ST1_ProductionDataValues:=	 CONCAT( ST1_ProductionDataValues,stStation1_ProductionData.DefaultNettWeight);
ST1_ProductionDataValues:= CONCAT( ST1_ProductionDataValues,',');
ST1_ProductionDataValues:=	 CONCAT( ST1_ProductionDataValues,stStation1_ProductionData.DefaultGrossWeight);
ST1_ProductionDataValues:= CONCAT( ST1_ProductionDataValues,',');
ST1_ProductionDataValues:=	 CONCAT( ST1_ProductionDataValues,stStation1_ProductionData.Blend);
ST1_ProductionDataValues:= CONCAT( ST1_ProductionDataValues,',');
ST1_ProductionDataValues:=	 CONCAT( ST1_ProductionDataValues,stStation1_ProductionData.Shade);
ST1_ProductionDataValues:= CONCAT( ST1_ProductionDataValues,',');
ST1_ProductionDataValues:=	 CONCAT( ST1_ProductionDataValues,stStation1_ProductionData.ConeTip);
ST1_ProductionDataValues:= CONCAT( ST1_ProductionDataValues,',');
ST1_ProductionDataValues:=	 CONCAT( ST1_ProductionDataValues,stStation1_ProductionData.ConeNettWeight);
ST1_ProductionDataValues:= CONCAT( ST1_ProductionDataValues,',');
ST1_ProductionDataValues:=	 CONCAT( ST1_ProductionDataValues,stStation1_ProductionData.ConeLength);
ST1_ProductionDataValues:= CONCAT( ST1_ProductionDataValues,',');
ST1_ProductionDataValues:=	 CONCAT( ST1_ProductionDataValues,stStation1_ProductionData.Dom_Exp);
ST1_ProductionDataValues:= CONCAT( ST1_ProductionDataValues,',');
ST1_ProductionDataValues:=	 CONCAT( ST1_ProductionDataValues,stStation1_ProductionData.PackType);
ST1_ProductionDataValues:= CONCAT( ST1_ProductionDataValues,',');
ST1_ProductionDataValues:=	 CONCAT( ST1_ProductionDataValues,stStation1_ProductionData.CountCode);
ST1_ProductionDataValues:= CONCAT( ST1_ProductionDataValues,'$0A');
(*==========Saving the Data to Report===========*)


sStation1_ProductionData_FileName:= Fb_CreateFileFormat_1.sOldFileName ; (*    'Hard Disk\Reports\Test1\ProductionData.csv' ;*)


Fb_LoagProductionData(
	bStartDataLog:= SaveData ,
	sDataLogFileName:=sStation1_ProductionData_FileName ,
	LogData:=ST1_ProductionDataValues ,
	bErrorDataLog=> );






(*=============== file copy from CX Controller to Remote PC & File Delete In CX Device======================*)


	Fb_CopyBackupAL_Server_LogOf_1(
		bMakeDirectory:= ,
		bCopyFile:=bool2,
		sDestDriveName:=' \\Admin-PC\Public\',
		sSourceDirectory:='\Hard Disk\Reports\Indo' ,
		 );

(*\\ramrajg-nb2\Ramaraj_public\   *)

  (*Hard Disk\Reports\  *)

Fb_FormatDrive_1(sDriveName:= '\\Admin-PC\Public\', bFormatDisk:=bFileDelete );

R_TRIG1(CLK:=CycleComplete OR CycleComplete1 , Q=> );


CASE ReportStep OF

	0:	 IF R_TRIG1.Q   THEN  FileCreateTemp:=TRUE; Timer3(IN:=FALSE); ReportStep:=1; END_IF

	1:	(*		##### Station 1 Production Data	#####	*)

		ST1_ProductionData:= CONCAT( 'S.No',',');
		ST1_ProductionData:=	 CONCAT( ST1_ProductionData,'Cone Type');
		ST1_ProductionData:= CONCAT( ST1_ProductionData,',');
		ST1_ProductionData:=	 CONCAT( ST1_ProductionData,'Carton No');
		ST1_ProductionData:= CONCAT( ST1_ProductionData,',');
		ST1_ProductionData:=	 CONCAT( ST1_ProductionData,'Lot No');
		ST1_ProductionData:= CONCAT( ST1_ProductionData,',');
		ST1_ProductionData:=	 CONCAT( ST1_ProductionData,'Date');
		ST1_ProductionData:= CONCAT( ST1_ProductionData,',');
		ST1_ProductionData:=	 CONCAT( ST1_ProductionData,'Net Weight');
		ST1_ProductionData:= CONCAT( ST1_ProductionData,',');
		ST1_ProductionData:=	 CONCAT( ST1_ProductionData,'Work Order No');
		ST1_ProductionData:= CONCAT( ST1_ProductionData,',');

ST1_ProductionData:=	 CONCAT( ST1_ProductionData,'Default Net Weight');
		ST1_ProductionData:= CONCAT( ST1_ProductionData,',');
ST1_ProductionData:=	 CONCAT( ST1_ProductionData,'Defaulr Gross Weight');
		ST1_ProductionData:= CONCAT( ST1_ProductionData,',');
ST1_ProductionData:=	 CONCAT( ST1_ProductionData,'Blend');
		ST1_ProductionData:= CONCAT( ST1_ProductionData,',');
ST1_ProductionData:=	 CONCAT( ST1_ProductionData,'Shade');
		ST1_ProductionData:= CONCAT( ST1_ProductionData,',');
ST1_ProductionData:=	 CONCAT( ST1_ProductionData,'Cone Tip');
		ST1_ProductionData:= CONCAT( ST1_ProductionData,',');
ST1_ProductionData:=	 CONCAT( ST1_ProductionData,'Cone Nett Weight');
		ST1_ProductionData:= CONCAT( ST1_ProductionData,',');
ST1_ProductionData:=	 CONCAT( ST1_ProductionData,'Cone Length');
		ST1_ProductionData:= CONCAT( ST1_ProductionData,',');
ST1_ProductionData:=	 CONCAT( ST1_ProductionData,'Dom Exp');
		ST1_ProductionData:= CONCAT( ST1_ProductionData,',');
ST1_ProductionData:=	 CONCAT( ST1_ProductionData,'Pack Type');
		ST1_ProductionData:=CONCAT( ST1_ProductionData,',');
ST1_ProductionData:=	 CONCAT( ST1_ProductionData,'CountCode');
		ST1_ProductionData:= CONCAT( ST1_ProductionData,'$0A');
		ReportStep:=2;

	2:	Timer1(IN:=FALSE);
		bANewDay:=FALSE;
		ReportStep:=3;


	3:	bEnableFileFormat:=TRUE;
		Timer1(IN:=TRUE , PT:=T#100ms , Q=> , ET=> );
		IF Timer1.Q THEN bEnableFileFormat:=FALSE;  ReportStep:=4; END_IF


	4:
		SaveData:=TRUE;
		Timer1(IN:=FALSE);
		ReportStep:=5;

	5:	Timer3(IN:=TRUE , PT:=T#25s , Q=> , ET=> );
		IF Timer3.Q THEN SaveData:=FALSE;bFileDelete:=TRUE; ReportStep:=6; END_IF

	6:	 bFileDelete:=FALSE;Timer3(IN:=FALSE); FileCreateTemp:=FALSE; ReportStep:=0;

END_CASE





IF ParametesSave THEN LotNoChange:=TRUE;ELSE LotNoChange:=FALSE;END_IF

IF bAutoModeOn AND bAPauseSeq AND   LotNoChange  THEN
	CurrentCartonNo:=CartonNoHmi;LotChangeCompleted:=FALSE;SameLotNo:=FALSE;
 END_IF

IF bAutoModeOn AND LotChangeCompleted THEN
	iLotNoPrevious:=iLotNoHmi;
END_IF



IF iLotNoPrevious=iLotNoHmi THEN SameLotNo:=TRUE;
ELSE SameLotNo:=FALSE;END_IF

CASE CartonNo OF

0: 	IF (CycleComplete OR CycleComplete1) THEN CartonNo:=CartonNo+1;TON_CountCheck(IN:=FALSE);END_IF

1:	IF SameLotNo THEN CartonNo:=CartonNo+1;
	ELSIF NOT SameLotNo THEN CartonNo:=3;END_IF

2:	CurrentCartonNo:=CurrentCartonNo+1;CartonNo:=4;

3:	CurrentCartonNo:=CartonNoHmi;CartonNo:=CartonNo+1;

4:	TON_CountCheck(IN:=TRUE, PT:=t#30s, Q=> , ET=> );
	IF TON_CountCheck.Q THEN CartonNo:=CartonNo+1;END_IF

5:	CartonNo:=0;LotChangeCompleted:=TRUE;

END_CASE









(*
CASE StepTemp1 OF
	0:	IF bRetUnitBStart THEN rRetUnitBWeightTemp1:=rRetUnitBWeight; StepTemp1:=StepTemp1+1; END_IF

	1:	IF UnitBCompleteCheckCount.CV = 18 AND bAutoModeOn THEN rRetUnitBWeightTemp2:=rRetUnitBWeightTemp1;  StepTemp1:=0; END_IF
 END_CASE




CASE StepTemp2 OF
	0:	IF bRetUnitBStart THEN rRetUnitBWeightTemp1:=rRetUnitBWeight; StepTemp2:=StepTemp2+1; END_IF

	1:	IF c18_ConeCounter1.CV = 18 AND bAutoModeOn THEN rRetUnitBWeightTemp2:=rRetUnitBWeightTemp1; c18_ConeCounter1.RESET:=TRUE;  StepTemp2:=StepTemp2+1; END_IF

	2:	c18_ConeCounter1.RESET:=FALSE;  StepTemp2:=0;
 END_CASE*)


(*IF LotAHmi AND NOT LotBHmi AND NOT LotCHmi THEN LotASelected:=TRUE;LotBSelected:=FALSE;LotCSelected:=FALSE;END_IF
IF NOT LotAHmi AND  LotBHmi AND NOT LotCHmi THEN LotBSelected:=TRUE;LotASelected:=FALSE;LotCSelected:=FALSE;END_IF
IF NOT LotAHmi AND NOT LotBHmi AND  LotCHmi THEN LotCSelected:=TRUE;LotBSelected:=FALSE;LotASelected:=FALSE;END_IF

IF LotASelected THEN CartonNoHmi:=LotACartonNo;
ELSIF LotBSelected THEN CartonNoHmi:=LotBCartonNo;
ELSIF  LotCSelected THEN CartonNoHmi:=LotCCartonNo;
ELSIF  LotDSelected THEN CartonNoHmi:=LotDCartonNo;
ELSIF  LotESelected THEN CartonNoHmi:=LotECartonNo;
ELSIF  LotFSelected THEN CartonNoHmi:=LotFCartonNo;
END_IF

IF CartonNoResetHmi OR  (NOT LotAHmi AND NOT LotBHmi AND NOT LotCHmi) THEN
	LotACartonNo:=0;
	LotBCartonNo:=0;
	LotCCartonNo:=0;
	LotDCartonNo:=0;
	LotECartonNo:=0;
	LotFCartonNo:=0;
END_IF



CASE LotA OF

0:	IF LotASelected THEN LotA:=LotA+1;END_IF

1:	IF (CycleComplete OR CycleComplete1) THEN LotA :=LotA +1;END_IF

2:	LotACartonNo:=LotACartonNo+1;
	LotA :=LotA +1;

3:	TON_11(IN:=TRUE , PT:=t#25s , Q=> , ET=> );
	IF TON_11.Q THEN LotA :=LotA +1;END_IF

4:	LotA :=0;

END_CASE


CASE LotB OF

0:	IF LotBSelected THEN LotB:=LotB+1;END_IF

1:	IF (CycleComplete OR CycleComplete1) THEN LotB:=LotB+1;END_IF

2:	LotBCartonNo:=LotBCartonNo+1;
	LotB:=LotB+1;

3:	TON_12(IN:=TRUE , PT:=t#25s , Q=> , ET=> );
	IF TON_12.Q THEN LotA :=LotA +1;END_IF

4:	LotB:=0;

END_CASE


CASE LotC OF

0:	IF LotCSelected THEN LotC:=LotC+1;END_IF

1:	IF (CycleComplete OR CycleComplete1) THEN LotC:=LotC+1;END_IF

2:	LotCCartonNo:=LotCCartonNo+1;
	LotC:=LotC+1;

3:	TON_13(IN:=TRUE , PT:=t#25s , Q=> , ET=> );
	IF TON_13.Q THEN LotA :=LotA +1;END_IF

4:	LotC:=0;

END_CASE*)
END_PROGRAM

(* POU FunctionBlocks/DATA_LOG_Save, ST *)
FUNCTION_BLOCK DATA_LOG_Save
VAR_INPUT
	bStartDataLog: BOOL;
	sDataLogFileName: STRING;
	LogData: STRING(1024);

END_VAR
VAR_OUTPUT

	bErrorDataLog: BOOL;
END_VAR
VAR

	R_TRIGStartDataLog: R_TRIG;
	nstep: INT;

	FB_OpenFile_Datalog: FB_FileOpen;
	nFB_OpenFile_Datalog_Errid: UDINT;

	FB_WriteFile_Datalog: FB_FileWrite;
	nFB_WriteFile_Datalog_ErrId: UDINT;

	FB_CloseFile_Datalog: FB_FileClose;
	nFB_CloseFile_Datalog_ErrId: UDINT;
	hDataLogSrcFile: UINT;

END_VAR
R_TRIGStartDataLog(CLK:=bStartDataLog , Q=> );
IF R_TRIGStartDataLog.Q THEN
		nstep :=1;
	END_IF

CASE nstep OF

	0:
		;
		FB_OpenFile_Datalog.bExecute:=FALSE;
		FB_WriteFile_Datalog.bExecute:=FALSE;
		FB_CloseFile_Datalog.bExecute:=FALSE;

	1:		(* do nothing *)
			nstep:=nstep+1;

	2:		(* ####	File Open ####*)

			FB_OpenFile_Datalog(  bExecute := FALSE  );
			FB_OpenFile_Datalog(	sNetId :='192.168.0.103.1.1' ,
			sPathName := sDataLogFileName,
			nMode := FOPEN_MODEAPPEND    ,
			ePath := PATH_GENERIC,
			tTimeout := T#2s,
			bExecute := TRUE );
			nstep := nstep+ 1;



	3:		FB_OpenFile_Datalog( bExecute := FALSE );
			IF ( NOT FB_OpenFile_Datalog.bBusy ) THEN
			IF ( FB_OpenFile_Datalog.bError ) THEN
			nFB_OpenFile_Datalog_Errid := FB_OpenFile_Datalog.nErrId;
			bErrorDataLog := TRUE;
			nstep := 50;
			ELSE
			hDataLogSrcFile := FB_OpenFile_Datalog.hFile;
			nstep := nstep + 1;
			END_IF
			END_IF

	4:		(*write data to destination file*)
			(*num:=num+1;*)
			FB_WriteFile_Datalog( bExecute := FALSE );
			FB_WriteFile_Datalog(	sNetId:='192.168.0.103.1.1',
			hFile:=FB_OpenFile_Datalog.hFile,
			pWriteBuff:= ADR(LogData),
			cbWriteLen:= LEN(LogData),		(*	i_len,	*)
			bExecute:=TRUE,
			tTimeout:=T#2s );
			nstep := nstep + 1;

	5:		FB_WriteFile_Datalog( bExecute := FALSE );
			IF ( NOT FB_WriteFile_Datalog.bBusy ) THEN
			IF ( FB_WriteFile_Datalog.bError ) THEN
			nFB_WriteFile_Datalog_ErrId := FB_WriteFile_Datalog.nErrId;
			bErrorDataLog := TRUE;
			nstep := 50;
			ELSE
			hDataLogSrcFile := FB_OpenFile_Datalog.hFile;
			nstep := nstep + 1;
			END_IF
			END_IF

	6:		(* close the destination file *)
			FB_CloseFile_Datalog( bExecute := FALSE );
			FB_CloseFile_Datalog( 	sNetId:='192.168.0.103.1.1' ,
			hFile:=FB_OpenFile_Datalog.hFile,
			bExecute:=TRUE,
			tTimeout:=T#2s );
			nstep := nstep + 1;

	7:		FB_CloseFile_Datalog( bExecute := FALSE );
			IF ( NOT FB_CloseFile_Datalog.bBusy ) THEN
			IF ( FB_CloseFile_Datalog.bError ) THEN
			nFB_CloseFile_Datalog_ErrId := FB_CloseFile_Datalog.nErrId;
			bErrorDataLog := TRUE;
			END_IF
			nstep := 0;
			END_IF

END_CASE
END_FUNCTION_BLOCK

(* POU FunctionBlocks/Fb_CreateFileFormat, LD *)
FUNCTION_BLOCK Fb_CreateFileFormat
VAR
	Fb_OpenFile: FB_FileOpen;
	Fb_WriteFile: FB_FileWrite;
	F_Trig1: F_TRIG;
	F_Trig2: F_TRIG;
	Fb_closeFile: FB_FileClose;
	F_Trig3: F_TRIG;


	SysteMtime: FB_LocalSystemTime;
	stSystemtimeAlrm: Timestruct;

	sFileName_Temp: T_MaxString;


	bCreateFileTrig: R_TRIG;
	bCreateFile: BOOL;
	Fb_SavePersistant: FB_WritePersistentData;
	TuneparaSave: BOOL;
END_VAR
VAR_INPUT

	sInputMessage: STRING(255);
	sFileName: T_MaxString;
	sDirectory: T_MaxString;
	bEnable: BOOL;

END_VAR
VAR_OUTPUT

	sDate: STRING;

	bNewDateFound: BOOL;
END_VAR

VAR_OUTPUT PERSISTENT
	sOldFileName: T_MaxString;
	sFilePathFinal: t_MaxString;
END_VAR
VAR PERSISTENT
	sOldDate: STRING;
	sNewFileName_Temp: T_MaxString;
END_VAR
VAR_IN_OUT PERSISTENT
	wToday: STRING;
END_VAR
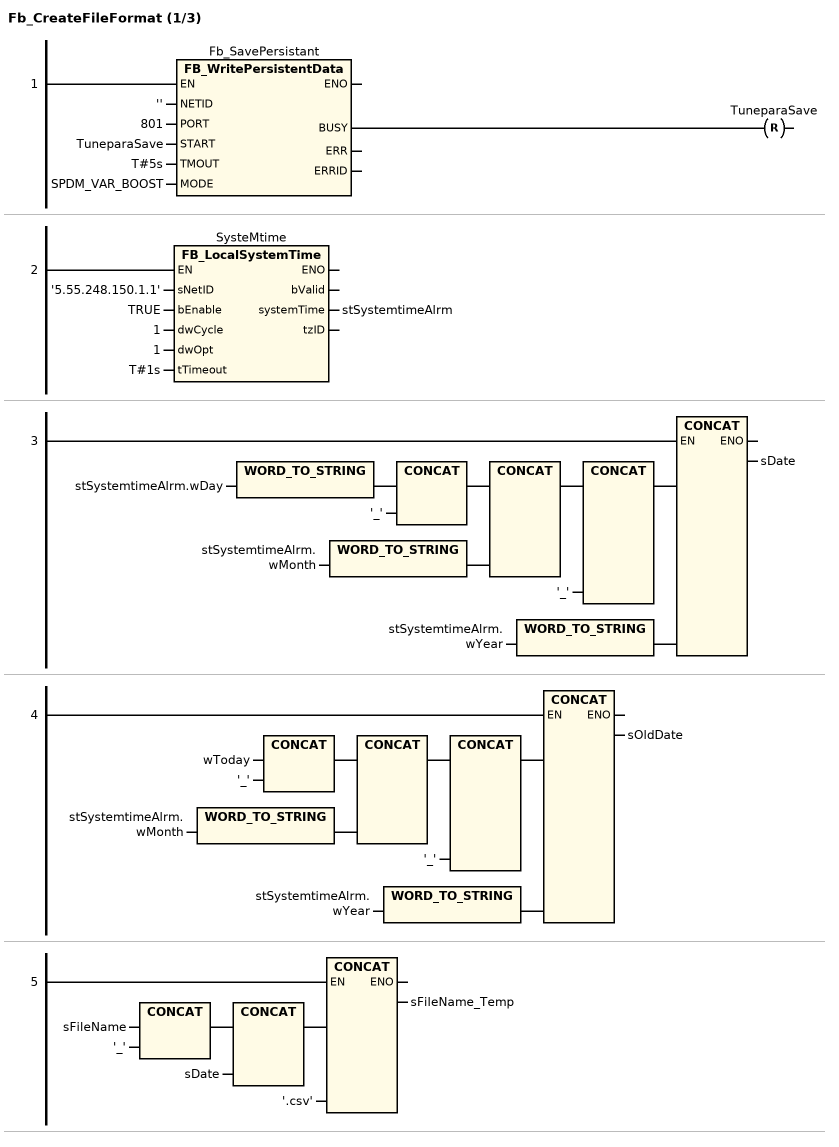
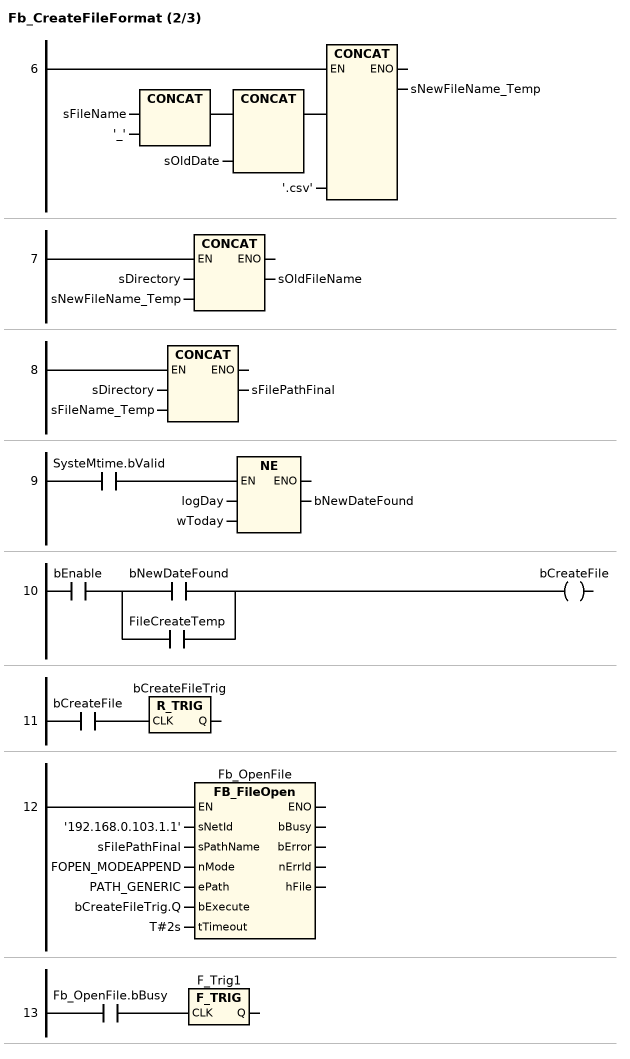
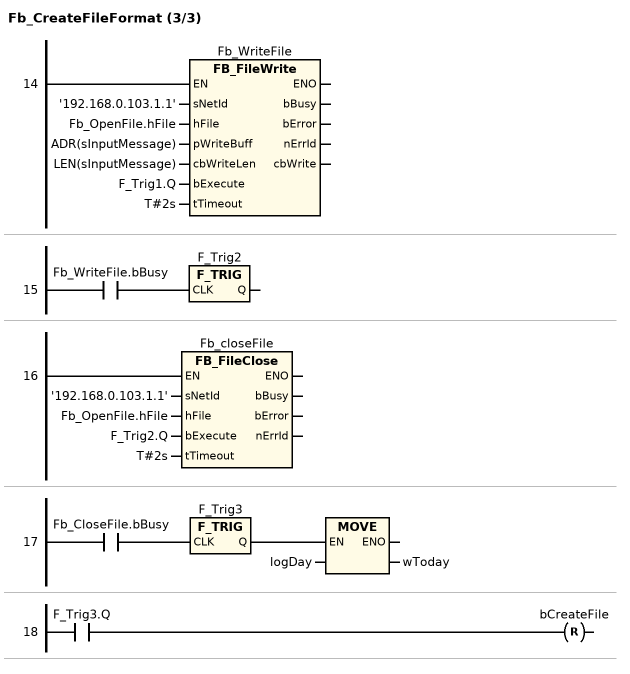
_LD_ (* Ladder Diagram *)
NETWORK 1
	*
		EN --- Fb_SavePersistant:FB_WritePersistentData(NETID: '', PORT: 801, START: TuneparaSave, TMOUT: T#5s, MODE: SPDM_VAR_BOOST) => R TuneparaSave
NETWORK 2
	*
		EN --- SysteMtime:FB_LocalSystemTime(sNetID: '5.55.248.150.1.1', bEnable: TRUE, dwCycle: 1, dwOpt: 1, tTimeout: T#1s, systemTime => stSystemtimeAlrm)
NETWORK 3
	*
		EN --- CONCAT(CONCAT(CONCAT(CONCAT(WORD_TO_STRING(stSystemtimeAlrm.wDay), '_'), WORD_TO_STRING(stSystemtimeAlrm.wMonth)), '_'), WORD_TO_STRING(stSystemtimeAlrm.wYear)) => sDate
NETWORK 4
	*
		EN --- CONCAT(CONCAT(CONCAT(CONCAT(wToday, '_'), WORD_TO_STRING(stSystemtimeAlrm.wMonth)), '_'), WORD_TO_STRING(stSystemtimeAlrm.wYear)) => sOldDate
NETWORK 5
	*
		EN --- CONCAT(CONCAT(CONCAT(sFileName, '_'), sDate), '.csv') => sFileName_Temp
NETWORK 6
	*
		EN --- CONCAT(CONCAT(CONCAT(sFileName, '_'), sOldDate), '.csv') => sNewFileName_Temp
NETWORK 7
	*
		EN --- CONCAT(sDirectory, sNewFileName_Temp) => sOldFileName
NETWORK 8
	*
		EN --- CONCAT(sDirectory, sFileName_Temp) => sFilePathFinal
NETWORK 9
	[SysteMtime.bValid]
		EN --- NE(logDay, wToday) => bNewDateFound
NETWORK 10
	[bEnable] - { [bNewDateFound] | [FileCreateTemp] } --- (bCreateFile)
NETWORK 11
	[bCreateFile] - bCreateFileTrig:R_TRIG(CLK: *)
NETWORK 12
	*
		EN --- Fb_OpenFile:FB_FileOpen(sNetId: '192.168.0.103.1.1', sPathName: sFilePathFinal, nMode: FOPEN_MODEAPPEND, ePath: PATH_GENERIC, bExecute: bCreateFileTrig.Q, tTimeout: T#2s)
NETWORK 13
	[Fb_OpenFile.bBusy] - F_Trig1:F_TRIG(CLK: *)
NETWORK 14
	*
		EN --- Fb_WriteFile:FB_FileWrite(sNetId: '192.168.0.103.1.1', hFile: Fb_OpenFile.hFile, pWriteBuff: ADR(sInputMessage), cbWriteLen: LEN(sInputMessage), bExecute: F_Trig1.Q, tTimeout: T#2s)
NETWORK 15
	[Fb_WriteFile.bBusy] - F_Trig2:F_TRIG(CLK: *)
NETWORK 16
	*
		EN --- Fb_closeFile:FB_FileClose(sNetId: '192.168.0.103.1.1', hFile: Fb_OpenFile.hFile, bExecute: F_Trig2.Q, tTimeout: T#2s)
NETWORK 17
	[Fb_CloseFile.bBusy] - F_Trig3:F_TRIG(CLK: *)
		EN --- MOVE(logDay) => wToday
NETWORK 18
	[F_Trig3.Q] --- (R bCreateFile)
_END_LD_
(* the same logic as Structured Text *)
(* Network 1 *)
Fb_SavePersistant(NETID := '', PORT := 801, START := TuneparaSave, TMOUT := T#5s, MODE := SPDM_VAR_BOOST);
IF Fb_SavePersistant.BUSY THEN TuneparaSave := FALSE; END_IF;
(* Network 2 *)
SysteMtime(sNetID := '5.55.248.150.1.1', bEnable := TRUE, dwCycle := 1, dwOpt := 1, tTimeout := T#1s);
stSystemtimeAlrm := SysteMtime.systemTime;
(* Network 3 *)
sDate := CONCAT(CONCAT(CONCAT(CONCAT(WORD_TO_STRING(stSystemtimeAlrm.wDay), '_'), WORD_TO_STRING(stSystemtimeAlrm.wMonth)), '_'), WORD_TO_STRING(stSystemtimeAlrm.wYear));
(* Network 4 *)
sOldDate := CONCAT(CONCAT(CONCAT(CONCAT(wToday, '_'), WORD_TO_STRING(stSystemtimeAlrm.wMonth)), '_'), WORD_TO_STRING(stSystemtimeAlrm.wYear));
(* Network 5 *)
sFileName_Temp := CONCAT(CONCAT(CONCAT(sFileName, '_'), sDate), '.csv');
(* Network 6 *)
sNewFileName_Temp := CONCAT(CONCAT(CONCAT(sFileName, '_'), sOldDate), '.csv');
(* Network 7 *)
sOldFileName := CONCAT(sDirectory, sNewFileName_Temp);
(* Network 8 *)
sFilePathFinal := CONCAT(sDirectory, sFileName_Temp);
(* Network 9 *)
IF SysteMtime.bValid THEN
	bNewDateFound := logDay <> wToday;
END_IF;
(* Network 10 *)
bCreateFile := bEnable AND (bNewDateFound OR FileCreateTemp);
(* Network 11 *)
bCreateFileTrig(CLK := bCreateFile);
(* Network 12 *)
Fb_OpenFile(sNetId := '192.168.0.103.1.1', sPathName := sFilePathFinal, nMode := FOPEN_MODEAPPEND, ePath := PATH_GENERIC, bExecute := bCreateFileTrig.Q, tTimeout := T#2s);
(* Network 13 *)
F_Trig1(CLK := Fb_OpenFile.bBusy);
(* Network 14 *)
Fb_WriteFile(sNetId := '192.168.0.103.1.1', hFile := Fb_OpenFile.hFile, pWriteBuff := ADR(sInputMessage), cbWriteLen := LEN(sInputMessage), bExecute := F_Trig1.Q, tTimeout := T#2s);
(* Network 15 *)
F_Trig2(CLK := Fb_WriteFile.bBusy);
(* Network 16 *)
Fb_closeFile(sNetId := '192.168.0.103.1.1', hFile := Fb_OpenFile.hFile, bExecute := F_Trig2.Q, tTimeout := T#2s);
(* Network 17 *)
F_Trig3(CLK := Fb_CloseFile.bBusy);
IF F_Trig3.Q THEN
	wToday := logDay;
END_IF;
(* Network 18 *)
IF F_Trig3.Q THEN bCreateFile := FALSE; END_IF;
END_FUNCTION_BLOCK

(* POU AutoMode/Fb_FormatDrive, FBD *)
FUNCTION_BLOCK Fb_FormatDrive
VAR_INPUT
	sDriveName: T_MaxString;
	bFormatDisk: BOOL;
END_VAR
VAR_OUTPUT
END_VAR
VAR
	sDeleteCommand_Temp: T_MaxString;
	sDeleteCommand: T_MaxString;
	nDirectoryLength: INT;
	sFormatedDirectory: T_MaxString;
	FbFormatDisk: NT_StartProcess;
END_VAR
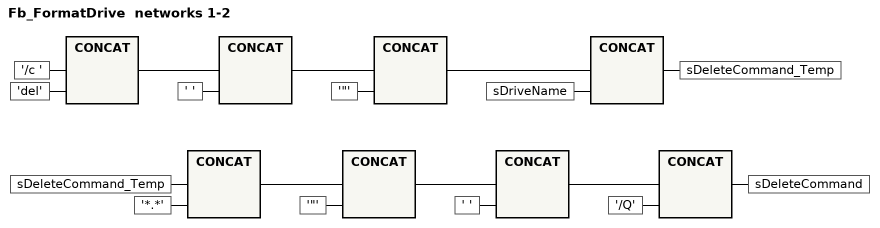
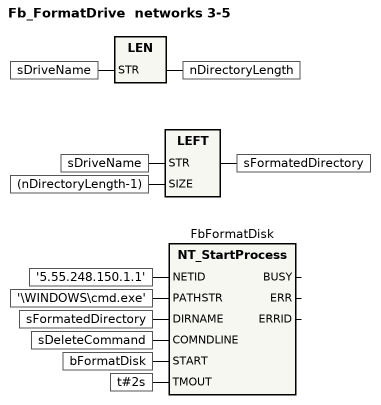
_FBD_ (* Function Block Diagram *)
NETWORK 1
	CONCAT(CONCAT(CONCAT(CONCAT('/c ', 'del'), ' '), '"'), sDriveName) => sDeleteCommand_Temp
NETWORK 2
	CONCAT(CONCAT(CONCAT(CONCAT(sDeleteCommand_Temp, '*.*'), '"'), ' '), '/Q') => sDeleteCommand
NETWORK 3
	LEN(STR: sDriveName) => nDirectoryLength
NETWORK 4
	LEFT(STR: sDriveName, SIZE: (nDirectoryLength-1)) => sFormatedDirectory
NETWORK 5
	FbFormatDisk:NT_StartProcess(NETID: '5.55.248.150.1.1', PATHSTR: '\WINDOWS\cmd.exe', DIRNAME: sFormatedDirectory, COMNDLINE: sDeleteCommand, START: bFormatDisk, TMOUT: t#2s)
_END_FBD_
(* the same logic as Structured Text *)
(* Network 1 *)
sDeleteCommand_Temp := CONCAT(CONCAT(CONCAT(CONCAT('/c ', 'del'), ' '), '"'), sDriveName);
(* Network 2 *)
sDeleteCommand := CONCAT(CONCAT(CONCAT(CONCAT(sDeleteCommand_Temp, '*.*'), '"'), ' '), '/Q');
(* Network 3 *)
nDirectoryLength := LEN(sDriveName);
(* Network 4 *)
sFormatedDirectory := LEFT(sDriveName, (nDirectoryLength-1));
(* Network 5 *)
FbFormatDisk(NETID := '5.55.248.150.1.1', PATHSTR := '\WINDOWS\cmd.exe', DIRNAME := sFormatedDirectory, COMNDLINE := sDeleteCommand, START := bFormatDisk, TMOUT := t#2s);
END_FUNCTION_BLOCK

(* POU FunctionBlocks/Fb_CopyFileToRemotePC, FBD *)
FUNCTION_BLOCK Fb_CopyFileToRemotePC
VAR
	sCopyFileCommandTemp: T_MaxString;
	sFormatedDestDirectory: T_Maxstring;
	sCopyFileCommand: T_MaxString;
	sFormatedDirectory: T_MaxString;
	sMakeDirCommand: T_MaxString;

	Fb_SystemTime: FB_LocalSystemTime;
	FB_MakeDirectory: NT_StartProcess;
	Fb_CopyFiles: NT_StartProcess;
END_VAR
VAR_INPUT

	bMakeDirectory: BOOL;
	bCopyFile: BOOL;
	sDestDriveName: T_MaxString;
	sSourceDirectory: T_MaxString;
END_VAR
VAR_OUTPUT
	sFinalDestDirectory: T_MaxString;
END_VAR
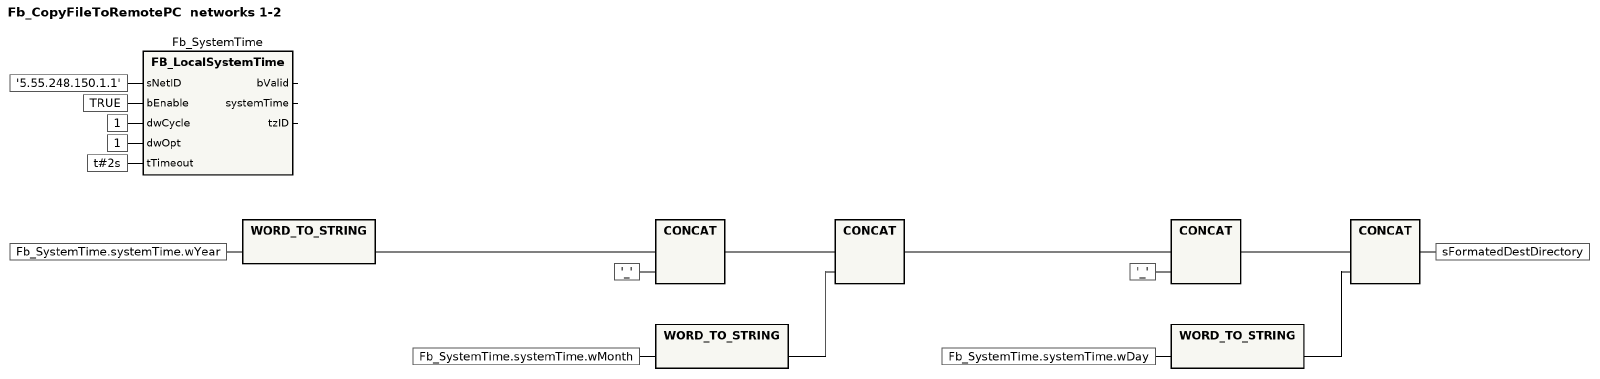
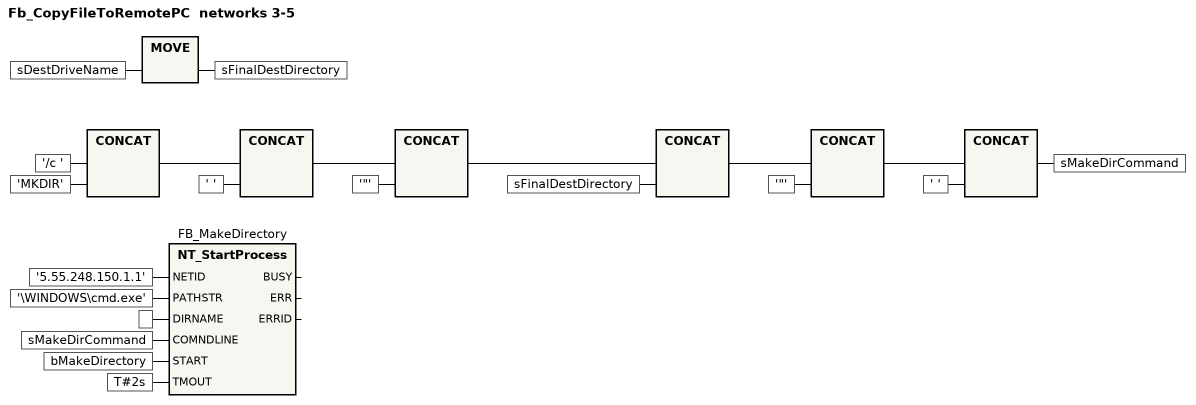
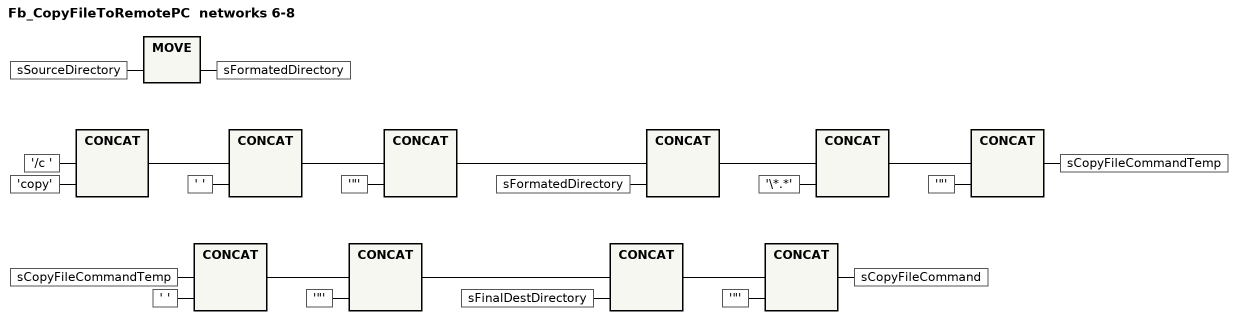
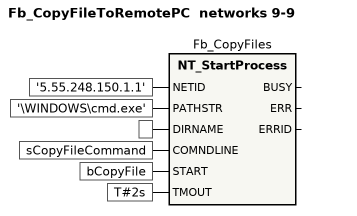
_FBD_ (* Function Block Diagram *)
NETWORK 1
	Fb_SystemTime:FB_LocalSystemTime(sNetID: '5.55.248.150.1.1', bEnable: TRUE, dwCycle: 1, dwOpt: 1, tTimeout: t#2s)
NETWORK 2
	CONCAT(CONCAT(CONCAT(CONCAT(WORD_TO_STRING(Fb_SystemTime.systemTime.wYear), '_'), WORD_TO_STRING(Fb_SystemTime.systemTime.wMonth)), '_'), WORD_TO_STRING(Fb_SystemTime.systemTime.wDay)) => sFormatedDestDirectory
NETWORK 3
	MOVE(sDestDriveName) => sFinalDestDirectory
NETWORK 4
	CONCAT(CONCAT(CONCAT(CONCAT(CONCAT(CONCAT('/c ', 'MKDIR'), ' '), '"'), sFinalDestDirectory), '"'), ' ') => sMakeDirCommand
NETWORK 5
	FB_MakeDirectory:NT_StartProcess(NETID: '5.55.248.150.1.1', PATHSTR: '\WINDOWS\cmd.exe', DIRNAME: , COMNDLINE: sMakeDirCommand, START: bMakeDirectory, TMOUT: T#2s)
NETWORK 6
	MOVE(sSourceDirectory) => sFormatedDirectory
NETWORK 7
	CONCAT(CONCAT(CONCAT(CONCAT(CONCAT(CONCAT('/c ', 'copy'), ' '), '"'), sFormatedDirectory), '\*.*'), '"') => sCopyFileCommandTemp
NETWORK 8
	CONCAT(CONCAT(CONCAT(CONCAT(sCopyFileCommandTemp, ' '), '"'), sFinalDestDirectory), '"') => sCopyFileCommand
NETWORK 9
	Fb_CopyFiles:NT_StartProcess(NETID: '5.55.248.150.1.1', PATHSTR: '\WINDOWS\cmd.exe', DIRNAME: , COMNDLINE: sCopyFileCommand, START: bCopyFile, TMOUT: T#2s)
_END_FBD_
(* the same logic as Structured Text *)
(* Network 1 *)
Fb_SystemTime(sNetID := '5.55.248.150.1.1', bEnable := TRUE, dwCycle := 1, dwOpt := 1, tTimeout := t#2s);
(* Network 2 *)
sFormatedDestDirectory := CONCAT(CONCAT(CONCAT(CONCAT(WORD_TO_STRING(Fb_SystemTime.systemTime.wYear), '_'), WORD_TO_STRING(Fb_SystemTime.systemTime.wMonth)), '_'), WORD_TO_STRING(Fb_SystemTime.systemTime.wDay));
(* Network 3 *)
sFinalDestDirectory := sDestDriveName;
(* Network 4 *)
sMakeDirCommand := CONCAT(CONCAT(CONCAT(CONCAT(CONCAT(CONCAT('/c ', 'MKDIR'), ' '), '"'), sFinalDestDirectory), '"'), ' ');
(* Network 5: see the listing above *)
(* Network 6 *)
sFormatedDirectory := sSourceDirectory;
(* Network 7 *)
sCopyFileCommandTemp := CONCAT(CONCAT(CONCAT(CONCAT(CONCAT(CONCAT('/c ', 'copy'), ' '), '"'), sFormatedDirectory), '\*.*'), '"');
(* Network 8 *)
sCopyFileCommand := CONCAT(CONCAT(CONCAT(CONCAT(sCopyFileCommandTemp, ' '), '"'), sFinalDestDirectory), '"');
(* Network 9: see the listing above *)
END_FUNCTION_BLOCK

(* Visualisation A
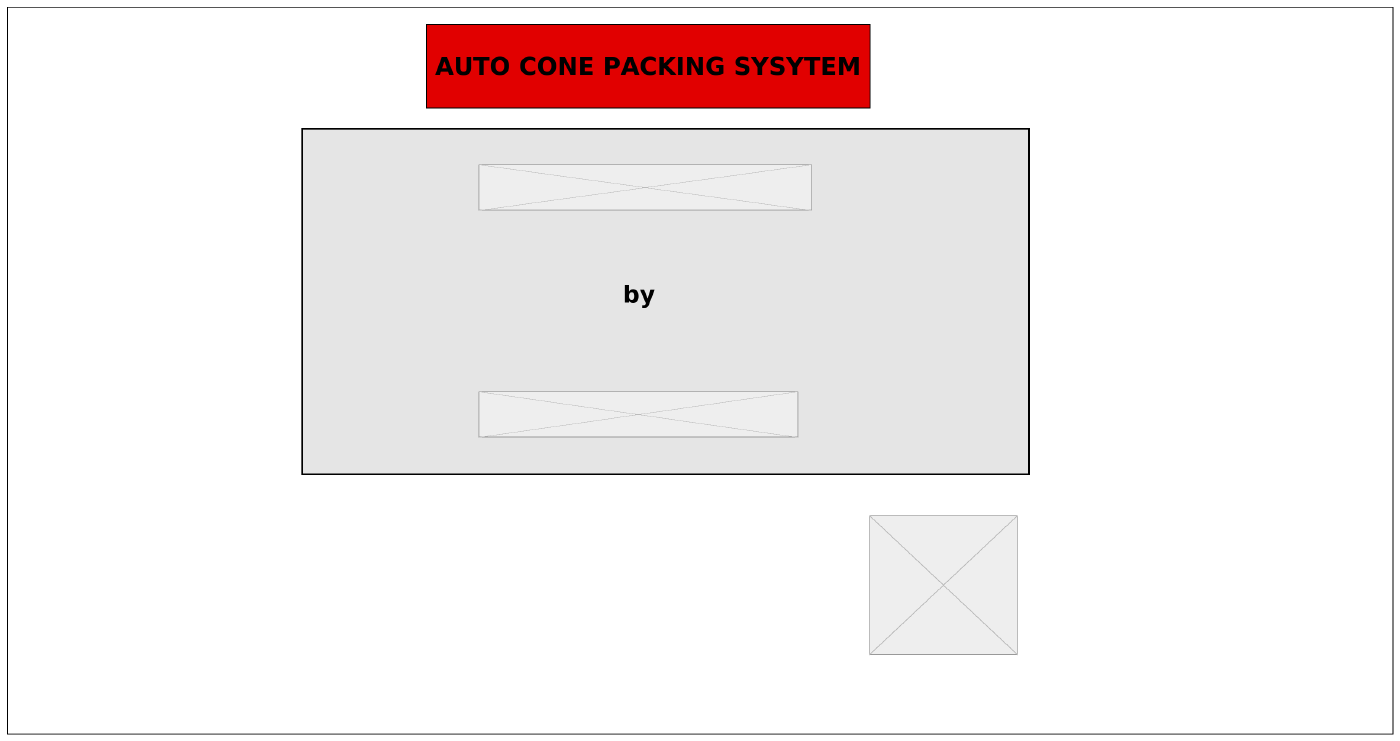
rounded rectangle at (484,20)-(997,117): text "AUTO CONE PACKING SYSYTEM"
bitmap at (996,588)-(1167,749): c:\twincat\plc\visu\startbutton.jpg
group at (340,140)-(1181,541)
  rounded rectangle at (0,0)-(1051,611): invisible if Common.EverRunTimer.Q
  bitmap at (256,64)-(737,145): c:\twincat\plc\visu\autocone-logom1.jpg
  bitmap at (256,464)-(717,545): c:\twincat\plc\visu\indo_logo1.bmp
  rectangle at (232,248)-(743,339): text "by"
2 more shapes without text or variables
*)

(* Visualisation ALARM
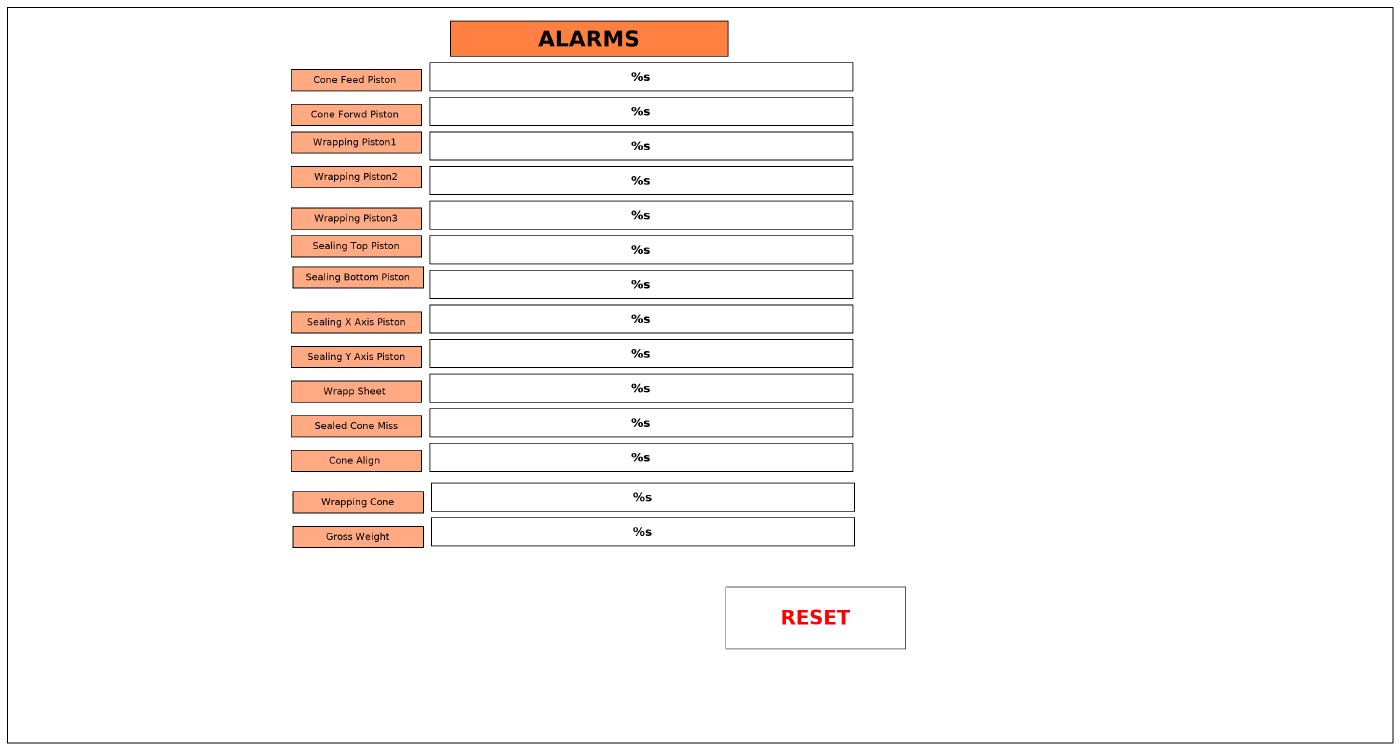
rounded rectangle at (328,112)-(479,137): text "Cone Forwd Piston"
rounded rectangle at (328,72)-(479,97): text "Cone Feed Piston"
rounded rectangle at (328,144)-(479,169): text "Wrapping Piston1"
rounded rectangle at (328,184)-(479,209): text "Wrapping Piston2"
rounded rectangle at (328,232)-(479,257): text "Wrapping Piston3"
rounded rectangle at (328,264)-(479,289): text "Sealing Top Piston"
rounded rectangle at (330,300)-(481,325): text "Sealing Bottom Piston"
rounded rectangle at (328,352)-(479,377): text "Sealing X Axis Piston"
rounded rectangle at (328,392)-(479,417): text "Sealing Y Axis Piston"
rectangle at (488,64)-(977,97): text "%s"; shows .HMIFeedPiston
rectangle at (488,224)-(977,257): text "%s"; shows .HMIWrapPiston3
rectangle at (488,184)-(977,217): text "%s"; shows .HMIWrapPiston2
rectangle at (488,264)-(977,297): text "%s"; shows .HMISealTopPiston
rectangle at (488,344)-(977,377): text "%s"; shows .HmiXAxisPiston
rectangle at (488,304)-(977,337): text "%s"; shows .HMISealBotPiston
rectangle at (488,384)-(977,417): text "%s"; shows .HmiYAxisPiston
rectangle at (488,144)-(977,177): text "%s"; shows .HMIWrapPiston1
rectangle at (488,104)-(977,137): text "%s"; shows .HMIForwdPiston
button at (830,670)-(1038,742): text "RESET"; shows .bErrorReset; taps .bErrorReset
rounded rectangle at (328,432)-(479,457): text "Wrapp Sheet"
rectangle at (488,424)-(977,457): text "%s"; shows ConeMissAlarm1
rounded rectangle at (328,472)-(479,497): text "Sealed Cone Miss"
rectangle at (488,464)-(977,497): text "%s"; shows .AlarmMessg
rounded rectangle at (328,512)-(479,537): text "Cone Align"
rectangle at (488,504)-(977,537): text "%s"; shows .ConeMissAlarm
rounded rectangle at (512,16)-(833,57): text "ALARMS"
rectangle at (490,550)-(979,583): text "%s"; shows WrapConeSenDetMes
rounded rectangle at (330,560)-(481,585): text "Wrapping Cone"
rectangle at (490,590)-(979,623): text "%s"; shows SGrossWtNokMsg
rounded rectangle at (330,600)-(481,625): text "Gross Weight"
1 more shapes without text or variables
2 elements of other kinds (tables, trends, ...) not read
*)

(* Visualisation ALARM_2
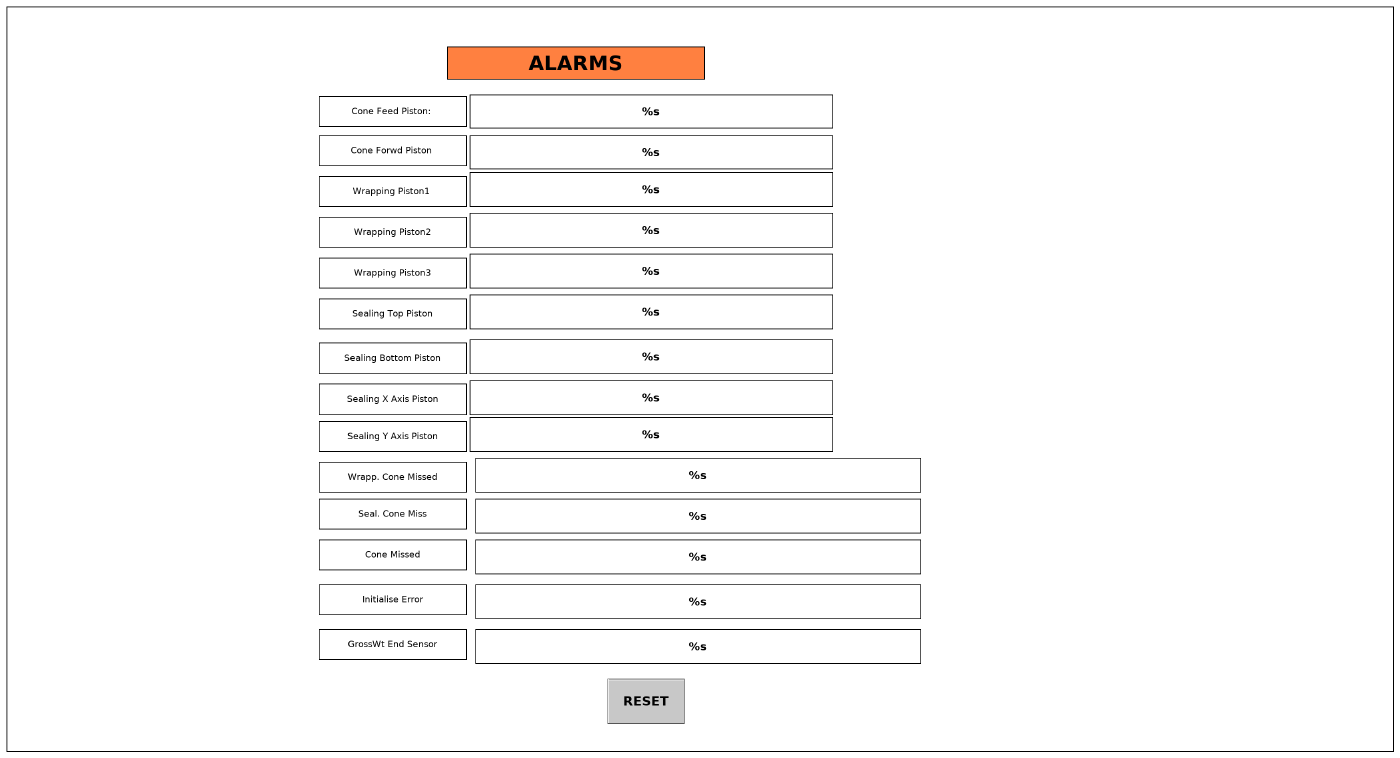
button at (750,830)-(846,886): text "RESET"; shows .bErrorReset; taps .bErrorReset
rounded rectangle at (550,40)-(871,81): text "ALARMS"
rounded rectangle at (390,151)-(574,189): text "Cone Forwd Piston"
rounded rectangle at (390,102)-(574,140): text "Cone Feed Piston:"
rounded rectangle at (390,202)-(574,240): text "Wrapping Piston1"
rounded rectangle at (390,253)-(574,291): text "Wrapping Piston2"
rounded rectangle at (390,304)-(574,342): text "Wrapping Piston3"
rounded rectangle at (390,355)-(574,393): text "Sealing Top Piston"
rounded rectangle at (390,410)-(574,449): text "Sealing Bottom Piston"
rounded rectangle at (390,461)-(574,500): text "Sealing X Axis Piston"
rounded rectangle at (390,508)-(574,546): text "Sealing Y Axis Piston"
rectangle at (578,100)-(1031,142): text "%s"; shows .HMIFeedPiston
rectangle at (578,299)-(1031,342): text "%s"; shows .HMIWrapPiston3
rectangle at (578,248)-(1031,291): text "%s"; shows .HMIWrapPiston2
rectangle at (578,350)-(1031,393): text "%s"; shows .HMISealTopPiston
rectangle at (578,457)-(1031,500): text "%s"; shows .HmiXAxisPiston
rectangle at (578,406)-(1031,449): text "%s"; shows .HMISealBotPiston
rectangle at (578,503)-(1031,546): text "%s"; shows .HmiYAxisPiston
rectangle at (578,197)-(1031,240): text "%s"; shows .HMIWrapPiston1
rectangle at (578,151)-(1031,193): text "%s"; shows .HMIForwdPiston
rounded rectangle at (390,559)-(574,597): text "Wrapp. Cone Missed"
rectangle at (585,554)-(1141,597): text "%s"; shows .ConeMissAlarm
rounded rectangle at (390,605)-(574,643): text "Seal. Cone Miss"
rectangle at (585,605)-(1141,648): text "%s"; shows .AlarmMessg
rounded rectangle at (390,656)-(574,694): text "Cone Missed"
rectangle at (585,656)-(1141,699): text "%s"; shows .ConeMissAlarm
rounded rectangle at (390,712)-(574,750): text "Initialise Error"
rectangle at (585,712)-(1141,755): text "%s"; shows sMessage
rounded rectangle at (390,768)-(574,806): text "GrossWt End Sensor"
rectangle at (585,768)-(1141,811): text "%s"; shows SGrossWtCylEndSenErrMsg
1 more shapes without text or variables
1 elements of other kinds (tables, trends, ...) not read
*)

(* Visualisation AUTO1
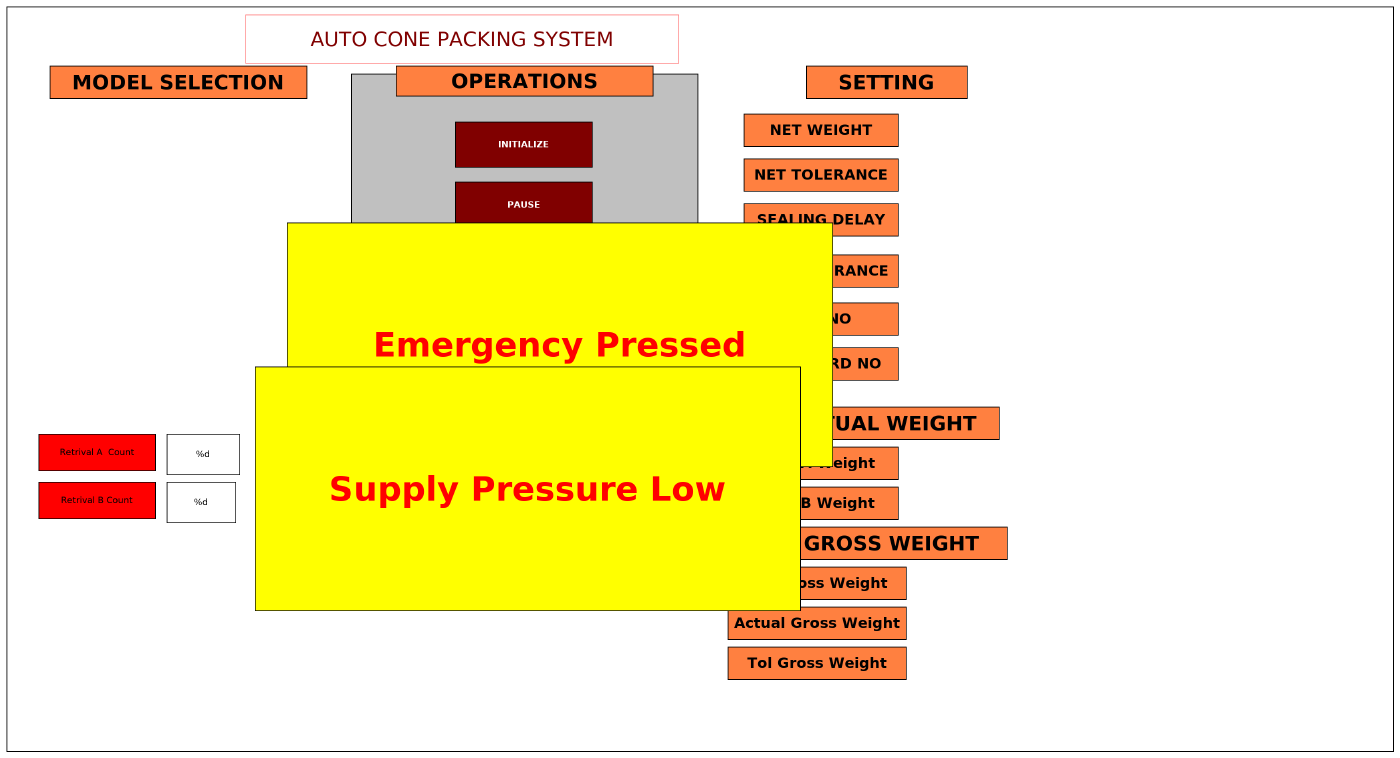
rounded rectangle at (298,10)-(839,71): text "AUTO CONE PACKING SYSTEM"
rounded rectangle at (326,538)-(527,579): text "Machine Status"
rounded rectangle at (542,530)-(855,587): text "%s"; shows sAMcModeStatus
rounded rectangle at (326,610)-(527,651): text "Alarm Status"
rounded rectangle at (542,602)-(855,659): text "%s"; shows sAlarmStatus
rounded rectangle at (54,74)-(375,115): text "MODEL SELECTION"
rounded rectangle at (920,550)-(1113,591): text "UnitA Weight"
rounded rectangle at (920,600)-(1113,641): text "UnitB Weight"
rounded rectangle at (920,246)-(1113,287): text "SEALING DELAY"
rounded rectangle at (998,74)-(1199,115): text "SETTING"
rounded rectangle at (920,134)-(1113,175): text "NET WEIGHT"
rounded rectangle at (920,190)-(1113,231): text "NET TOLERANCE"
rounded rectangle at (950,500)-(1239,541): text "ACTUAL WEIGHT"
rounded rectangle at (920,310)-(1113,351): text "NEG TOLERANCE"
rounded rectangle at (200,594)-(286,645): text "%d"; shows UnitBConeCountHMI
rounded rectangle at (200,534)-(291,585): text "%d"; shows UnitAConeCountHMI
rectangle at (40,534)-(186,580): text "Retrival A  Count"
rectangle at (40,594)-(186,640): text "Retrival B Count"
group at (430,74)-(863,494)
  rounded rectangle at (130,304)-(301,362): text "STOP"; alarm colour if bStopHmi; taps bStopHmi
  rounded rectangle at (130,221)-(301,279): text "RESUME"; alarm colour if bAPauseSeq; taps bResumeHmi
  rounded rectangle at (130,145)-(301,203): text "PAUSE"; alarm colour if bAPauseSeq; taps bPauseHmi
  rounded rectangle at (130,70)-(301,127): text "INITIALIZE"; alarm colour if bAInitializeSeq; taps bInitializeHmi
  rounded rectangle at (56,0)-(377,38): text "OPERATIONS"
rounded rectangle at (920,370)-(1113,411): text "LOT NO"
rounded rectangle at (900,700)-(1123,741): text "Set Gross Weight"
rounded rectangle at (900,750)-(1123,791): text "Actual Gross Weight"
rounded rectangle at (960,650)-(1249,691): text "GROSS WEIGHT"
rounded rectangle at (900,800)-(1123,841): text "Tol Gross Weight"
rounded rectangle at (920,426)-(1113,467): text "WORK ORD NO"
rounded rectangle at (350,270)-(1031,575): text "Emergency Pressed"; invisible if NOT bEmPopUp
rounded rectangle at (310,450)-(991,755): text "Supply Pressure Low"; invisible if NOT bPrssurePopUp
2 more shapes without text or variables
22 elements of other kinds (tables, trends, ...) not read
*)

(* Visualisation DIAGNOSTICS
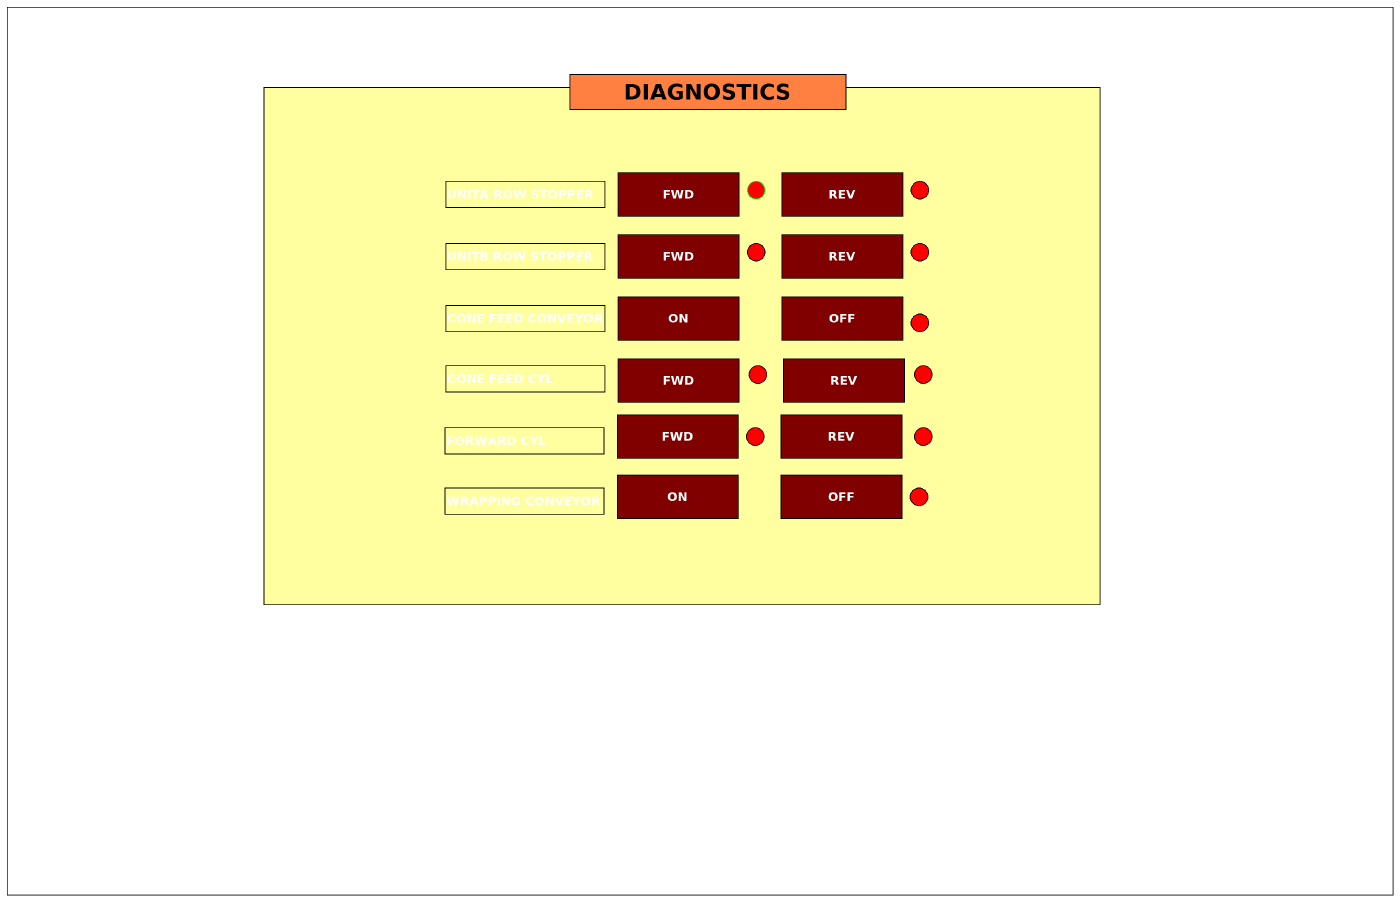
rounded rectangle at (645,70)-(966,111): text "DIAGNOSTICS"
ellipse at (851,194)-(872,215): alarm colour if .bIUnitA_RowStopperEnd
ellipse at (851,266)-(872,287): alarm colour if .bIUnitB_RowStopperEnd
ellipse at (1041,194)-(1062,215): alarm colour if .bIUnitA_RowStopperHome
ellipse at (1041,266)-(1062,287): alarm colour if .bIUnitB_RowStopperHome
ellipse at (1041,348)-(1062,369): alarm colour if .bQFeedingConveyorMotor
rounded rectangle at (701,184)-(842,235): text "FWD"; alarm colour if .bUA_RowStopperMotorFwdOnHmi; taps .bUA_RowStopperMotorFwdOnHmi
rounded rectangle at (891,184)-(1032,235): text "REV"; alarm colour if .bUA_RowStopperMotorRevOnHmi; taps .bUA_RowStopperMotorRevOnHmi
rounded rectangle at (701,256)-(842,307): text "FWD"; alarm colour if .bUB_RowStopperMotorFwdOnHmi; taps .bUB_RowStopperMotorFwdOnHmi
rounded rectangle at (701,328)-(842,379): text "ON"; alarm colour if bFCMotorOnHmi; taps bFCMotorOnHmi
rounded rectangle at (891,256)-(1032,307): text "REV"; alarm colour if .bUB_RowStopperMotorRevOnHmi; taps .bUB_RowStopperMotorRevOnHmi
rounded rectangle at (891,328)-(1032,379): text "OFF"; alarm colour if bFCMotorOffHmi; taps bFCMotorOffHmi
rounded rectangle at (501,194)-(686,225): text "UNITA ROW STOPPER"
rounded rectangle at (501,266)-(686,297): text "UNITB ROW STOPPER"
rounded rectangle at (501,338)-(686,369): text "CONE FEED CONVEYOR"
ellipse at (853,408)-(874,429): alarm colour if .bIConeFeedingPistonEnd
ellipse at (1045,408)-(1066,429): alarm colour if .bIConeFeedingPistonHome
rounded rectangle at (701,400)-(842,451): text "FWD"; alarm colour if .bCFPistonOnHmi; taps .bCFPistonOnHmi
rounded rectangle at (893,400)-(1034,451): text "REV"; alarm colour if .bCFPistonOffHmi; taps .bCFPistonOffHmi
rounded rectangle at (501,408)-(686,439): text "CONE FEED CYL"
ellipse at (1040,550)-(1061,571): alarm colour if .bQMWrappingConveyorMotor
rounded rectangle at (700,535)-(841,586): text "ON"; alarm colour if .bWCMotorOnHmi; taps .bWCMotorOnHmi
rounded rectangle at (890,535)-(1031,586): text "OFF"; alarm colour if .bWCMotorOffHmi; taps .bWCMotorOffHmi
rounded rectangle at (500,550)-(685,581): text "WRAPPING CONVEYOR"
rounded rectangle at (500,480)-(685,511): text "FORWARD CYL"
rounded rectangle at (700,465)-(841,516): text "FWD"; alarm colour if .bFPValveOnHmi; taps .bFPValveOnHmi
rounded rectangle at (890,465)-(1031,516): text "REV"; alarm colour if .bFPValveOffHmi; taps .bFPValveOffHmi
ellipse at (850,480)-(871,501): alarm colour if .bIForwardPistonEnd
ellipse at (1045,480)-(1066,501): alarm colour if .bIForwardPistonHome
2 more shapes without text or variables
2 elements of other kinds (tables, trends, ...) not read
*)

(* Visualisation DIAGNOSTICS_1
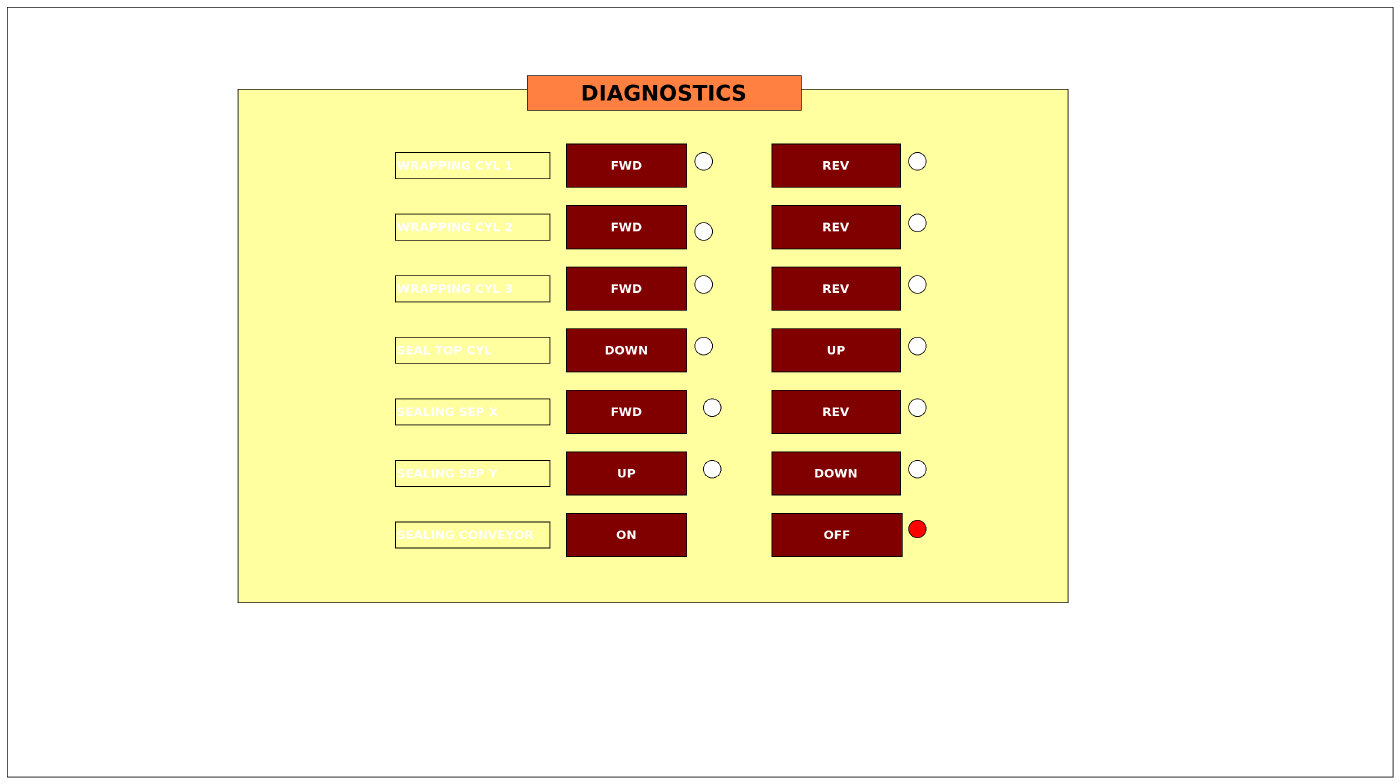
rounded rectangle at (608,80)-(929,121): text "DIAGNOSTICS"
rounded rectangle at (654,160)-(795,211): text "FWD"; alarm colour if .bWrappingCPV1OnHmi; taps .bWrappingCPV1OnHmi
rounded rectangle at (654,232)-(795,283): text "FWD"; alarm colour if .bWrappingCPV2OnHmi; taps .bWrappingCPV2OnHmi
rounded rectangle at (894,232)-(1045,283): text "REV"; alarm colour if .bWrappingCPV2OffHmi; taps .bWrappingCPV2OffHmi
rounded rectangle at (654,304)-(795,355): text "FWD"; alarm colour if .bWrappingCPV3OnHmi; taps .bWrappingCPV3OnHmi
rounded rectangle at (894,304)-(1045,355): text "REV"; alarm colour if .bWrappingCPV3OffHmi; taps .bWrappingCPV3OffHmi
rounded rectangle at (654,376)-(795,427): text "DOWN"; alarm colour if .bSealingTopPVOnHmi; taps .bSealingTopPVOnHmi
rounded rectangle at (894,376)-(1045,427): text "UP"; alarm colour if bSealingTopPVOffHmi; taps bSealingTopPVOffHmi
rounded rectangle at (654,448)-(795,499): text "FWD"; alarm colour if bSSXAxisPistonValveOnHmi; taps bSSXAxisPistonValveOnHmi
rounded rectangle at (894,448)-(1045,499): text "REV"; alarm colour if bSSXAxisPistonValveOffHmi; taps bSSXAxisPistonValveOffHmi
rounded rectangle at (454,170)-(635,201): text "WRAPPING CYL 1"
rounded rectangle at (454,242)-(635,273): text "WRAPPING CYL 2"
rounded rectangle at (454,314)-(635,345): text "WRAPPING CYL 3"
rounded rectangle at (454,386)-(635,417): text "SEAL TOP CYL"
rounded rectangle at (454,458)-(635,489): text "SEALING SEP X"
rounded rectangle at (894,160)-(1045,211): text "REV"; alarm colour if .bWrappingCPV1OffHmi; taps .bWrappingCPV1OffHmi
ellipse at (1054,600)-(1075,621): alarm colour if .bQMWrappingConveyorMotor
rounded rectangle at (654,592)-(795,643): text "ON"; alarm colour if bSCMotorOnHmi; taps bSCMotorOnHmi
rounded rectangle at (894,592)-(1047,643): text "OFF"; alarm colour if bSCMotorOffHmi; taps bSCMotorOffHmi
rounded rectangle at (454,602)-(635,633): text "SEALING CONVEYOR"
rounded rectangle at (654,520)-(795,571): text "UP"; alarm colour if bSSYAxisPistonValveOnHmi; taps bSSYAxisPistonValveOnHmi
rounded rectangle at (894,520)-(1045,571): text "DOWN"; alarm colour if bSSYAxisPistonValveOffHmi; taps bSSYAxisPistonValveOffHmi
rounded rectangle at (454,530)-(635,561): text "SEALING SEP Y"
14 more shapes without text or variables
2 elements of other kinds (tables, trends, ...) not read
*)

(* Visualisation OVERVIEW
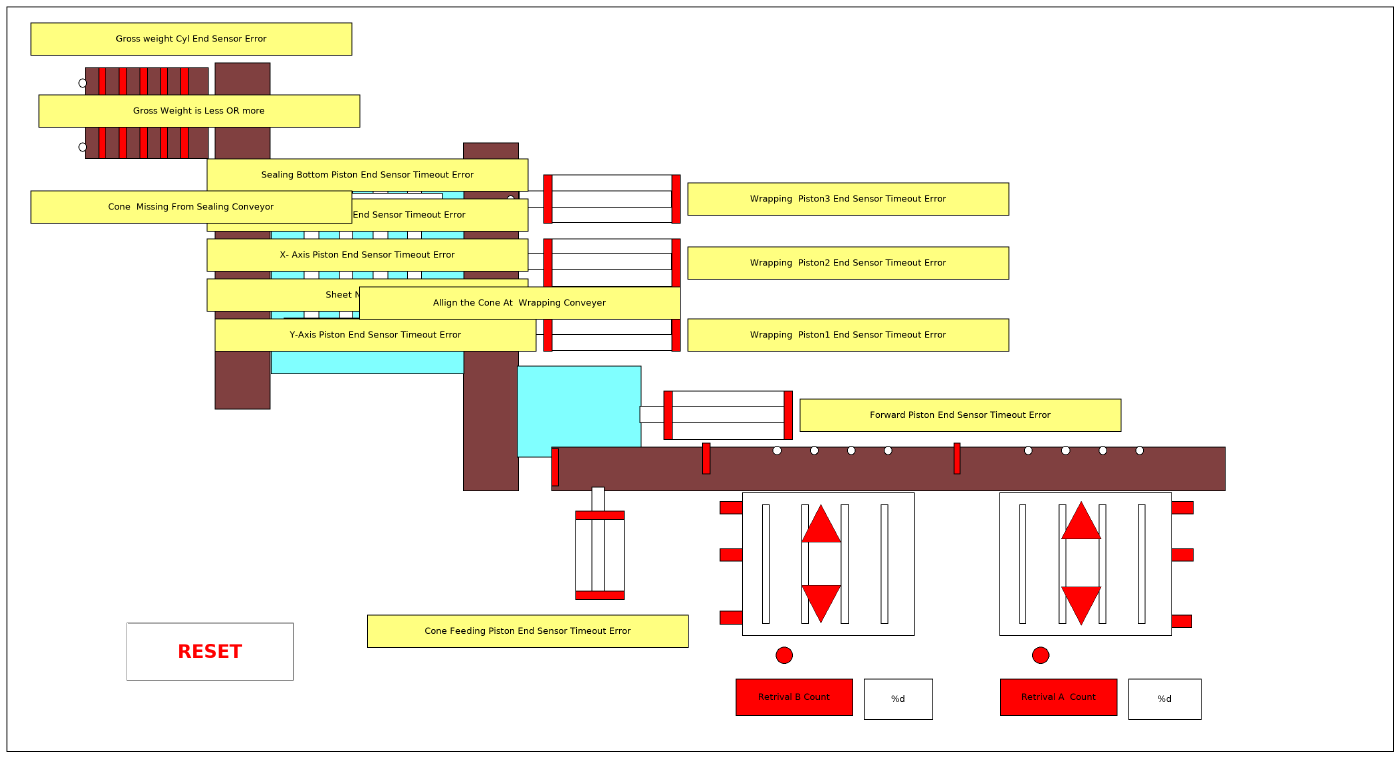
rectangle at (640,308)-(830,329): alarm colour if bQWrappingChannelPistonValve2
rectangle at (830,290)-(841,351): alarm colour if bIWrappingChannelPiston2_Home
rectangle at (1440,760)-(1479,776): alarm colour if bIUnitA_RowStopperHome
rectangle at (1446,677)-(1481,693): alarm colour if bIUnitA_RowStopperMiddle
rectangle at (1446,618)-(1481,634): alarm colour if bIUnitA_RowStopperEnd
rectangle at (890,618)-(922,634): alarm colour if bIUnitB_RowStopperEnd
rectangle at (890,755)-(922,772): alarm colour if bIUnitB_RowStopperHome
rectangle at (890,677)-(922,693): alarm colour if bIUnitB_RowStopperMiddle
rounded rectangle at (570,170)-(639,605): alarm colour if bQWrappingConveyorMotor
rectangle at (790,499)-(979,520): alarm colour if bQForwardPistonValve
rounded rectangle at (680,550)-(1521,605): alarm colour if bQFeedingConveyorMotor
polygon at (992,723)-(1041,770): alarm colour if bQUnitBRowStopperMotorRev
polygon at (992,622)-(1041,669): alarm colour if bQUnitBRowStopperMotorFwd
polygon at (1316,725)-(1366,773): alarm colour if bQUnitARowStopperMotorRev
polygon at (1316,618)-(1366,665): alarm colour if bQUnitARowStopperMotorFwd
rectangle at (680,552)-(689,599): alarm colour if bIConeOrientationTop
rectangle at (868,545)-(878,584): alarm colour if bIUnitBConeCrossing
rectangle at (1182,545)-(1190,584): alarm colour if bIUnitAConeCrossing
rectangle at (730,600)-(746,740): alarm colour if bQConeFeedingPistonValve
rectangle at (640,390)-(830,410): alarm colour if bQWrappingChannelPistonValve1
rectangle at (640,230)-(830,251): alarm colour if bQWrappingChannelPistonValve3
rectangle at (415,206)-(432,416): alarm colour if bQSealingBottomPistonValve
rectangle at (371,206)-(390,416): alarm colour if bQSealingSeparatorXAxisPistonValve
rectangle at (457,206)-(476,416): alarm colour if bQSealingTopPistonValve
rectangle at (500,210)-(518,421): alarm colour if bQSealingSeparatorYAxisPistonValve
rounded rectangle at (260,70)-(329,503): alarm colour if bQSealingConveyorMotorFWD
rectangle at (98,76)-(252,190): alarm colour if bQGross_Cylinder_On
rectangle at (192,76)-(201,190): alarm colour if bQGross_Roller_On
rectangle at (217,76)-(227,190): alarm colour if bQGross_Roller_On
rectangle at (166,76)-(176,190): alarm colour if bQGross_Roller_On
rectangle at (140,76)-(150,190): alarm colour if bQGross_Roller_On
rectangle at (115,76)-(124,190): alarm colour if bQGross_Roller_On
rectangle at (346,389)-(544,407): alarm colour if bQFilmRollerMotor1
rectangle at (346,233)-(544,250): alarm colour if bQFilmRollerMotor3
rectangle at (346,310)-(544,329): alarm colour if bQFilmRollerMotor2
ellipse at (1316,549)-(1327,560): alarm colour if bIUnitAConeDetection3
ellipse at (1363,549)-(1373,560): alarm colour if bIUnitAConeDetection2
ellipse at (1409,549)-(1419,560): alarm colour if bIUnitAConeDetection1
ellipse at (1270,549)-(1280,560): alarm colour if bIUnitAConeDetection4
ellipse at (1003,549)-(1013,560): alarm colour if bIUnitBConeDetection3
ellipse at (1049,549)-(1059,560): alarm colour if bIUnitBConeDetection2
ellipse at (1095,549)-(1105,560): alarm colour if bIUnitBConeDetection1
ellipse at (956,549)-(967,560): alarm colour if bIUnitBConeDetection4
ellipse at (624,236)-(634,247): alarm colour if bIWrappingCone3
ellipse at (624,314)-(634,325): alarm colour if bIWrappingCone2
ellipse at (620,390)-(630,401): alarm colour if bIWrappingCone1
ellipse at (283,197)-(293,207): alarm colour if bIConeCountSensor
ellipse at (513,190)-(523,200): alarm colour if bISealingSeparatorYAxisEnd
ellipse at (380,190)-(391,200): alarm colour if bISealingSeparatorXAxisEnd
ellipse at (476,190)-(486,200): alarm colour if bISealingTopPistonEnd
ellipse at (430,190)-(440,200): alarm colour if bISealingBottomPistonEnd
ellipse at (90,90)-(100,101): alarm colour if bIGross_Cyl_Home
ellipse at (90,170)-(100,181): alarm colour if bIGross_Cyl_End
ellipse at (960,800)-(981,821): alarm colour if bQUnitBWeightOkLamp
ellipse at (1280,800)-(1301,821): alarm colour if bQUnitAWeightOkLamp
rectangle at (830,210)-(841,271): alarm colour if bIWrappingChannelPiston3_Home
rectangle at (830,370)-(841,431): alarm colour if bIWrappingChannelPiston1_Home
rectangle at (710,630)-(771,641): alarm colour if bIConeFeedingPistonEnd
rectangle at (710,730)-(771,741): alarm colour if bIConeFeedingPistonHome
rectangle at (970,480)-(981,541): alarm colour if bIForwardPistonHome
ellipse at (509,420)-(520,431): alarm colour if bISealingSeparatorYAxisHome
ellipse at (380,420)-(390,431): alarm colour if bISealingSeparatorXAxisHome
ellipse at (472,420)-(483,431): alarm colour if bISealingTopPistonHome
ellipse at (426,420)-(436,431): alarm colour if bISealingBottomPistonHome
rectangle at (450,760)-(851,801): text "Cone Feeding Piston End Sensor Timeout Error"; invisible if NOT bAConeFeedCylRsError
rectangle at (850,390)-(1251,431): text "Wrapping  Piston1 End Sensor Timeout Error"; invisible if NOT bAWrappingCylRs1Error
rectangle at (850,220)-(1251,261): text "Wrapping  Piston3 End Sensor Timeout Error"; invisible if NOT bAWrappingCylRs3Error
rectangle at (850,300)-(1251,341): text "Wrapping  Piston2 End Sensor Timeout Error"; invisible if NOT bAWrappingCylRs2Error
rectangle at (250,190)-(651,231): text "Sealing Bottom Piston End Sensor Timeout Error"; invisible if NOT bASealBotCylRsError
rectangle at (250,240)-(651,281): text "Sealing Top Piston End Sensor Timeout Error"; invisible if NOT bASealTopCylRsError
rectangle at (250,290)-(651,331): text "X- Axis Piston End Sensor Timeout Error"; invisible if NOT bASealSepXCylRsError
rectangle at (260,390)-(661,431): text "Y-Axis Piston End Sensor Timeout Error"; invisible if NOT bASealSepYCylRsError
rectangle at (250,340)-(651,381): text "Sheet NOT Feeded"; invisible if NOT bAPolythinSheetError
rectangle at (30,230)-(431,271): text "Cone  Missing From Sealing Conveyor"; invisible if NOT bAConeMissAtSealConv
rectangle at (440,350)-(841,391): text "Allign the Cone At  Wrapping Conveyer"; invisible if NOT bAConeMissErrorAtWrpConv
rectangle at (40,110)-(441,151): text "Gross Weight is Less OR more"; invisible if NOT bGrossWieghtNOk
rectangle at (990,490)-(1391,531): text "Forward Piston End Sensor Timeout Error"; invisible if NOT bAFwdCylRsError
rectangle at (30,20)-(431,61): text "Gross weight Cyl End Sensor Error"; invisible if NOT bGrossWtCylEndSenError
button at (150,770)-(358,842): text "RESET"; shows .bErrorReset; taps .bErrorReset
rounded rectangle at (1070,840)-(1156,891): text "%d"; shows UnitBConeCountHMI
rounded rectangle at (1400,840)-(1491,891): text "%d"; shows UnitAConeCountHMI
rectangle at (1240,840)-(1386,886): text "Retrival A  Count"
rectangle at (910,840)-(1056,886): text "Retrival B Count"
22 more shapes without text or variables
6 elements of other kinds (tables, trends, ...) not read
*)

(* Visualisation PARAMETERS
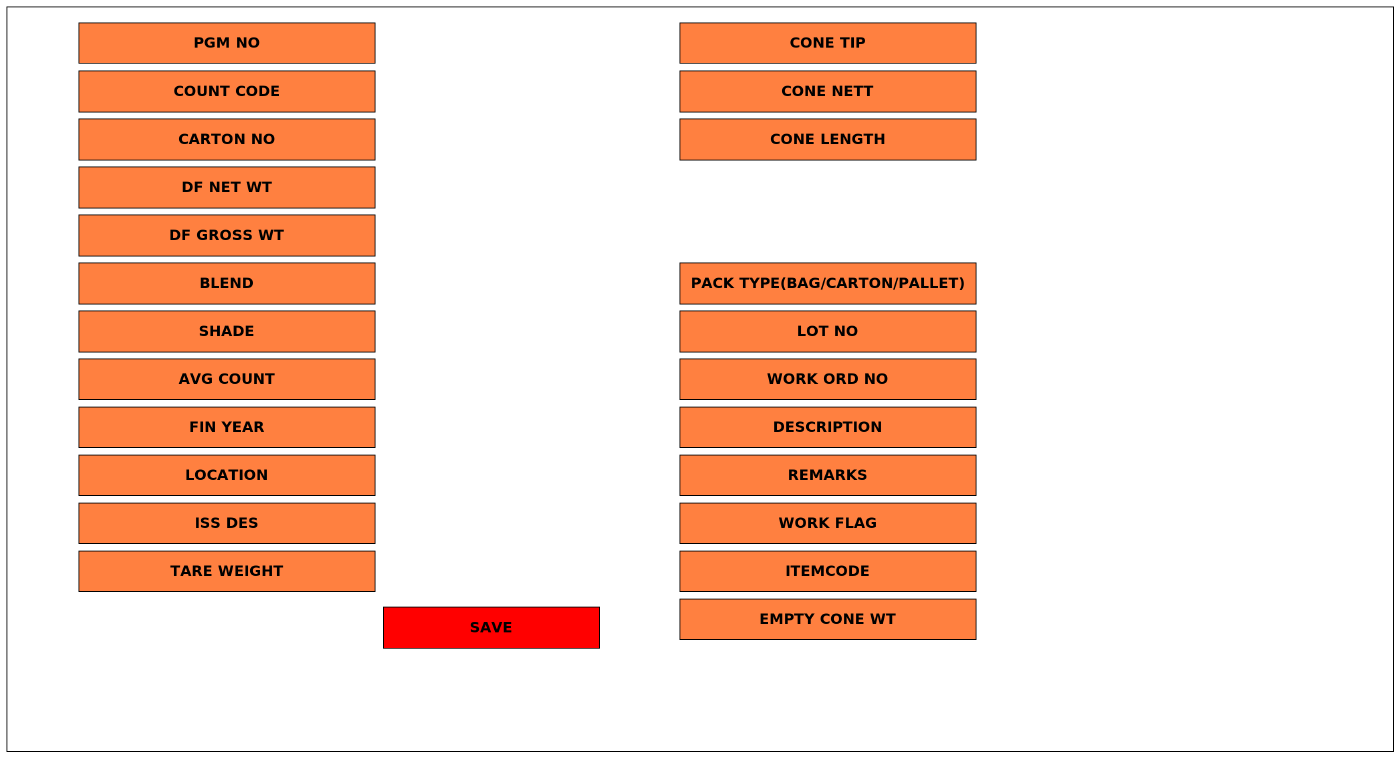
rounded rectangle at (90,20)-(460,71): text "PGM NO"
rounded rectangle at (90,80)-(460,132): text "COUNT CODE"
rounded rectangle at (90,200)-(460,252): text "DF NET WT"
rounded rectangle at (90,140)-(460,192): text "CARTON NO"
rounded rectangle at (90,260)-(460,312): text "DF GROSS WT"
rounded rectangle at (90,320)-(460,372): text "BLEND"
rounded rectangle at (90,380)-(460,432): text "SHADE"
rounded rectangle at (840,20)-(1210,71): text "CONE TIP"
rounded rectangle at (840,80)-(1210,132): text "CONE NETT"
rounded rectangle at (840,140)-(1210,192): text "CONE LENGTH"
rounded rectangle at (840,320)-(1210,372): text "PACK TYPE(BAG/CARTON/PALLET)"
rounded rectangle at (840,380)-(1210,432): text "LOT NO"
rounded rectangle at (840,440)-(1210,491): text "WORK ORD NO"
rounded rectangle at (470,750)-(740,802): text "SAVE"; alarm colour if ParametesSave; taps ParametesSave
rounded rectangle at (90,440)-(460,491): text "AVG COUNT"
rounded rectangle at (90,500)-(460,551): text "FIN YEAR"
rounded rectangle at (90,560)-(460,611): text "LOCATION"
rounded rectangle at (90,620)-(460,671): text "ISS DES"
rounded rectangle at (90,680)-(460,731): text "TARE WEIGHT"
rounded rectangle at (840,500)-(1210,551): text "DESCRIPTION"
rounded rectangle at (840,560)-(1210,611): text "REMARKS"
rounded rectangle at (840,620)-(1210,671): text "WORK FLAG"
rounded rectangle at (840,680)-(1210,731): text "ITEMCODE"
rounded rectangle at (840,740)-(1210,791): text "EMPTY CONE WT"
1 more shapes without text or variables
30 elements of other kinds (tables, trends, ...) not read
*)

(* Visualisation PARAMETERS_SAVE
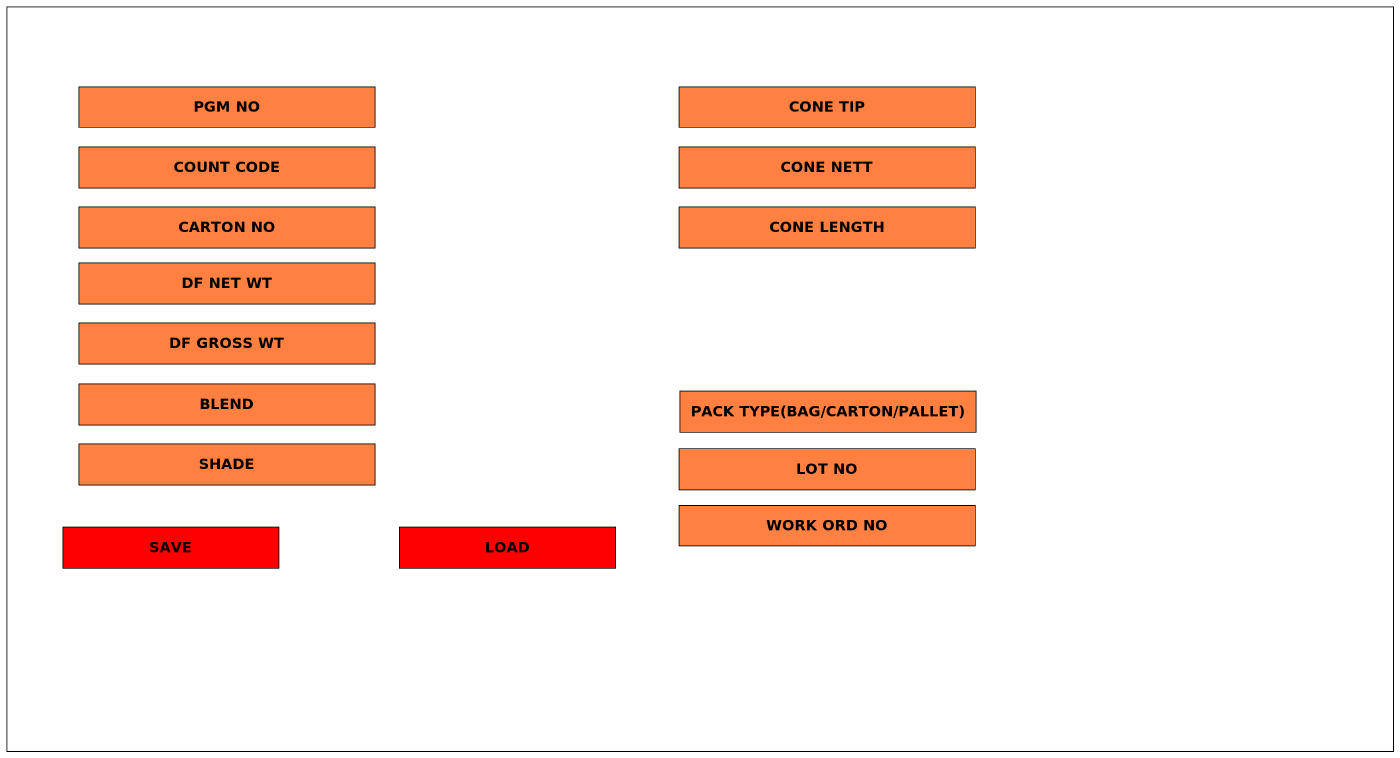
rounded rectangle at (100,110)-(470,161): text "PGM NO"
rounded rectangle at (100,185)-(470,237): text "COUNT CODE"
rounded rectangle at (100,330)-(470,382): text "DF NET WT"
rounded rectangle at (100,260)-(470,312): text "CARTON NO"
rounded rectangle at (100,405)-(470,457): text "DF GROSS WT"
rounded rectangle at (100,481)-(470,533): text "BLEND"
rounded rectangle at (100,556)-(470,608): text "SHADE"
rounded rectangle at (849,110)-(1219,161): text "CONE TIP"
rounded rectangle at (849,185)-(1219,237): text "CONE NETT"
rounded rectangle at (849,260)-(1219,312): text "CONE LENGTH"
rounded rectangle at (850,490)-(1220,542): text "PACK TYPE(BAG/CARTON/PALLET)"
rounded rectangle at (849,562)-(1219,614): text "LOT NO"
rounded rectangle at (849,633)-(1219,684): text "WORK ORD NO"
rounded rectangle at (80,660)-(350,712): text "SAVE"; alarm colour if SAVE; taps SAVE
rounded rectangle at (500,660)-(770,712): text "LOAD"; alarm colour if LOAD; taps LOAD
1 more shapes without text or variables
21 elements of other kinds (tables, trends, ...) not read
*)
